FUNCTION_BLOCK SEL_SENS (* Basic Function Block Type *)
  (* Standard: 61499-2 *)
  (* Version 0.2, 2003-12-04, JHC, Rockwell Automation, Renamed for better indexing. *)
  (* Version 0.1, 2002-11-05, JHC, Rockwell Automation, Corrected missing ST element in Algorithm REQ. *)
  (* Version 0.0, 2000-05-30, JHC, Rockwell Automation *)
  (* Compiler header: package fb.rt.vhmi; *)
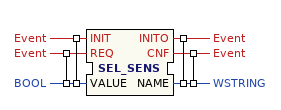
  EVENT_INPUT
    INIT WITH VALUE; (* Initialization Request *)
    REQ WITH VALUE; (* Normal Execution Request *)
  END_EVENT
  EVENT_OUTPUT
    INITO WITH NAME; (* Initialization Confirm *)
    CNF WITH NAME; (* Execution Confirmation *)
  END_EVENT
  VAR_INPUT
    VALUE : BOOL; (* Input event qualifier *)
  END_VAR
  VAR_OUTPUT
    NAME : WSTRING; (* Output event qualifier *)
  END_VAR
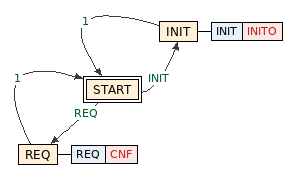
  EC_STATES
    START; (* Initial State *)
    INIT : INIT -> INITO; (* Initialization *)
    REQ : REQ -> CNF; (* Normal execution *)
  END_STATES
  EC_TRANSITIONS
    START TO INIT := INIT;
    INIT TO START := 1;
    START TO REQ := REQ;
    REQ TO START := 1;
  END_TRANSITIONS
  ALGORITHM INIT IN ST: (* Initialization algorithm *)
NAME:="/fb/rt/vhmi/sens0.gif";
  END_ALGORITHM
  ALGORITHM REQ IN ST: (* Normally executed algorithm *)
IF (VALUE=false) THEN NAME:="/fb/rt/vhmi/sens0.gif"; END_IF
IF (VALUE=true) THEN NAME:="/fb/rt/vhmi/sens1.gif"; END_IF
  END_ALGORITHM
END_FUNCTION_BLOCK
